FUNCTION_BLOCK FB_Alarm
VAR_INPUT
	AL_H1 : BOOL;	
	AL_H1_V : BOOL;
	AL_H2 : BOOL;
	AL_H2_V : BOOL;
	AL_H4 : BOOL;
	AL_H4_V : BOOL;
	Al_Sim : BOOL;
	T_Alarm : TIME;
	reset : BOOL;
END_VAR
VAR_OUTPUT
	GL_Alarm : BOOL;
END_VAR
VAR
	has_Alarm : BOOL;
	Alarm_On : TOF;
	Trig : F_TRIG;
	Alarm : RS;
END_VAR

has_Alarm := 
	AL_H1 OR 
	AL_H2 OR 
	AL_H4 OR 
	AL_H1_V OR 
	AL_H2_V OR 
	AL_H4_V OR
	AL_Sim;
	
Alarm_On(IN := has_Alarm, PT := T_Alarm);
TRIG(CLK := Alarm_On.Q);
Alarm(SET := has_Alarm, RESET1 :=  TRIG.Q OR reset, Q1 => GL_Alarm);

END_FUNCTION_BLOCK

(* stored: Version 1.1.0.1, ProductVersion 3.1.4018.5
   POU FB_Alarm: Id {572deef5-61f9-4ec5-93f6-0c170029445b}, SpecialFunc None *)
